FUNCTION convertToAm : REAL
VAR_INPUT
	pCommand	:	REAL;
	enaPosDir	:	BOOL;
END_VAR
VAR
END_VAR

//	0 to 1000 mA conversion
IF  enaPosDir THEN
	convertToAm:= (ABS(pCommand) * (generalVariable.conParammetr.CurPosDirMax - generalVariable.conParammetr.CurPosDirMin)/1000) + generalVariable.conParammetr.CurPosDirMin;
	ELSE
		convertToAm:= (ABS(pCommand) * (generalVariable.conParammetr.CurNegDirMax - generalVariable.conParammetr.CurNegDirMin)/1000) + generalVariable.conParammetr.CurNegDirMin;
		END_IF;

END_FUNCTION

(* stored: Version 1.1.0.1, ProductVersion 3.1.4024.12
   POU convertToAm: Id {a6c875f3-dbd7-4260-9c4b-f101c22c557f}, SpecialFunc None *)
